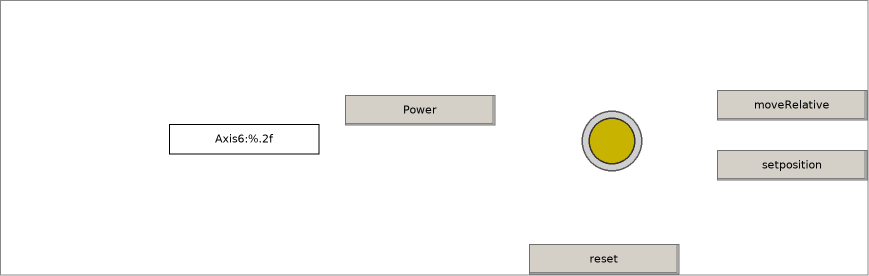
VISUALIZATION HMI  // 869x276
    Rectangle (169,124 150x30), "Axis6:%.2f", text variable: MAIN.axis6.NcToPlc.ActPos
    Button (345,95 150x30), "Power"
        toggle MAIN.power_do
    Lamp1 (577,106 70x70), variable: MAIN.axis6.NcToPlc.StateDWord.20, style: Lamp-Lamp1-Yellow
    Button (717,90 150x30), "moveRelative"
        tap MAIN.move_do
    Button (717,150 150x30), "setposition"
        tap MAIN.set_do
    Button (529,244 150x30), "reset"
        tap MAIN.reset_do
END_VISUALIZATION

(* stored: Version 1.1.0.1, ProductVersion 3.1.4022.16
   Visu HMI: Id {0f96c8bb-599b-4474-ac66-8fee7836104c} *)
